Universal Robots PolyScope program: run_driver.urp

Program run_driver (installation=default directory=/programs/usbdisk/script_driver createdIn=5.2.0.61336 lastSavedIn=5.3.0.64176 robotSerialNumber=20195000535)
Calibrated DH parameters: a=[0.000149, -0.595503, -0.570094, 0.000069, 0.000037, 0]; d=[0.180711, 684.397239, -686.764447, 2.541569, 0.119967, 0.115293]; alpha=[1.570175, 0.000207, -0.013852, 1.571079, -1.570194, 0]; deltaTheta=[0, 0.233602, -0.176156, -0.057447, 0, 0]
BeforeStart
  Script file /programs/usbdisk/script_driver/driver.script
    | def driver():
    |   # Initialize variables hi
    |   global mode_thread_running = -1
    |   reset_vars()
    |   # Setup thread to read and update registers
    |   run read_and_update()
    |   # Continuously run command() function, which handles running correct mode thread. The mode threads then command the robot.
    |   while (True):
    |     command()
    |     sync()
    |   end
    | end
    | 
    | def command():
    |   # Run correct mode thread, then continuously check if the current thread is still running.
    |   # If mode switches while a mode thread is currently running, kill that mode thread
    |   # Break the loop and return from this function once either the mode thread finishes or the mode thread is killed
    |   mode_thread_switch() # Run the correct mode thread. This will update global variable mode_thread_running
    |   sync()
    |   while (mode_thread_running != -1): # mode_thread_running = mode number of mode thread that is currently running, otherwise if no mode thread is running, it = -1
    |     if mode != mode_thread_running: # If mode switched while another mode thread is already running, kill the current mode thread before breaking loop
    |       kill mode_thread_handler
    |       mode_thread_running = -1
    |     else:
    |       sync()
    |     end
    |   end
    | end
    | 
    | def mode_thread_switch():
    |   # Based on current value of mode, run the corresponding mode thread
    |   end_freedrive_mode() # End freedrive mode (if not in freedrive mode, does nothing) before running a mode thread
    |   if mode == STANDBY_MODE or enable == 0:
    |     global mode_thread_handler = run standby()
    |   elif mode == FREEDRIVE_MODE:
    |     global mode_thread_handler = run freedrive()
    |   elif mode == WAYPOINT_JOINT_MODE:
    |     global mode_thread_handler = run waypointJoint()
    |   elif mode == WAYPOINT_CARTESIAN_MODE:
    |     global mode_thread_handler = run waypointCartesian()
    |   elif mode == POSITION_CONTROL_JOINT_MODE:
    |     global mode_thread_handler = run posControlJoint()
    |   elif mode == POSITION_CONTROL_CARTESIAN_MODE:
    |     global mode_thread_handler = run posControlCartesian()
    |   elif mode == VELOCITY_CONTROL_JOINT_MODE:
    |     global mode_thread_handler = run velControlJoint()
    |   elif mode == VELOCITY_CONTROL_CARTESIAN_MODE:
    |     global mode_thread_handler = run velControlCartesian()
    |   end
    | end
    | 
    | thread read_and_update():
    |   # Continuously
    |   while(True):
    |     write_output_integer_register(PING_OUTPUT_INT_REGISTER, read_input_integer_register(PING_INT_REGISTER))
    |     if mode != read_input_integer_register(MODE_INT_REGISTER): # If mode changed, reset variables and re-setup watchdogs
    |       reset_vars()
    |       mode = read_input_integer_register(MODE_INT_REGISTER)
    |       setup_watchdogs()
    |     end
    |     # Update each variable only if mode requires it to be updated. Create list of all modes which require variable to be updated and use list_contains() to check if current mode is one of those modes
    |     if list_contains(mode, [WAYPOINT_JOINT_MODE, WAYPOINT_CARTESIAN_MODE, POSITION_CONTROL_JOINT_MODE, POSITION_CONTROL_CARTESIAN_MODE, VELOCITY_CONTROL_JOINT_MODE, VELOCITY_CONTROL_CARTESIAN_MODE]):
    |       setp = read_registers_into_list(SETP_DOUBLE_REGISTER_OFFSET, 6, "DOUBLE")
    |     end
    |     if list_contains(mode, [WAYPOINT_JOINT_MODE, WAYPOINT_CARTESIAN_MODE,VELOCITY_CONTROL_JOINT_MODE]):
    |       avtr = read_registers_into_list(AVTR_DOUBLE_REGISTER_OFFSET, 4, "DOUBLE")
    |     end
    |     if list_contains(mode, [POSITION_CONTROL_JOINT_MODE, POSITION_CONTROL_CARTESIAN_MODE, VELOCITY_CONTROL_CARTESIAN_MODE]):
    |       servoj_params = read_registers_into_list(SERVOJ_PARAMS_DOUBLE_REGISTER_OFFSET, 3, "DOUBLE")
    |     end
    |     enable = read_input_integer_register(ENABLE_INT_REGISTER) # Always update enable regardless of mode
    |     sync()
    |   end
    | end
    | 
    | def reset_vars():
    |   global mode = 0
    |   global enable = 0
    |   global setp = [0.0,0.0,0.0,0.0,0.0,0.0]
    |   global avtr = [0.0,0.0,0.0,0.0]
    |   global servoj_params = [0.0,0.0,0.0]
    | end
    | 
    | def setup_watchdogs():
    |   # Depending on current mode, set watchdog frequencies and responses for each watchdog
    |   # Right now, frequency always set to 500Hz and response is "STOP" if mode requires that variable, or "IGNORE" otherwise
    |   # "STOP" preferred over "PAUSE" initially for safety. Once we are more comfortable with system, can use "PAUSE" where appropriate
    | 
    |   mode_freq = 1
    |   enable_freq = 1
    |   setp_freq = 1
    |   avtr_freq = 1
    |   servoj_params_freq = 1
    | 
    |   mode_resp = "IGNORE"
    |   enable_resp = "IGNORE"
    |   setp_resp = "IGNORE"
    |   avtr_resp = "IGNORE"
    |   servoj_params_resp = "IGNORE"
    | 
    |   if list_contains(mode, [POSITION_CONTROL_JOINT_MODE, POSITION_CONTROL_CARTESIAN_MODE, VELOCITY_CONTROL_JOINT_MODE, VELOCITY_CONTROL_CARTESIAN_MODE, FORCE_CONTROL_MODE]):
    |     mode_resp = "STOP"
    |   end
    |   if list_contains(mode, [POSITION_CONTROL_JOINT_MODE, POSITION_CONTROL_CARTESIAN_MODE, VELOCITY_CONTROL_JOINT_MODE, VELOCITY_CONTROL_CARTESIAN_MODE, FORCE_CONTROL_MODE]):
    |     enable_resp = "STOP"
    |   end
    |   if list_contains(mode, [POSITION_CONTROL_JOINT_MODE, POSITION_CONTROL_CARTESIAN_MODE, VELOCITY_CONTROL_JOINT_MODE, VELOCITY_CONTROL_CARTESIAN_MODE, FORCE_CONTROL_MODE]):
    |     setp_resp = "STOP"
    |   end
    |   if list_contains(mode, []):
    |     avtr_resp = "STOP"
    |   end
    |   if list_contains(mode, [POSITION_CONTROL_JOINT_MODE, POSITION_CONTROL_CARTESIAN_MODE, VELOCITY_CONTROL_CARTESIAN_MODE]):
    |     servoj_params_resp = "STOP"
    |   end
    | 
    |   rtde_set_watchdog("input_int_register_"+to_str(MODE_INT_REGISTER), mode_freq, mode_resp)
    |   rtde_set_watchdog("input_int_register_"+to_str(ENABLE_INT_REGISTER), enable_freq, enable_resp)
    |   rtde_set_watchdog("input_double_register_"+to_str(SETP_DOUBLE_REGISTER_OFFSET), setp_freq, setp_resp)
    |   rtde_set_watchdog("input_double_register_"+to_str(AVTR_DOUBLE_REGISTER_OFFSET), avtr_freq, avtr_resp)
    |   rtde_set_watchdog("input_double_register_"+to_str(SERVOJ_PARAMS_DOUBLE_REGISTER_OFFSET), servoj_params_freq, servoj_params_resp)
    | end
    | 
    | 
    | # MODE THREADS
    | # FIRST set mode_thread_running to the corresponding mode number.
    | # THEN body of thread
    | thread standby():
    |   mode_thread_running = STANDBY_MODE
    |   write_output_integer_register(MODE_OUTPUT_INT_REGISTER, mode_thread_running)
    |   while(True):
    |     if not is_steady():
    |       stopj(DEFAULT_JOINT_ACCELERATION)
    |     end
    |     sync()
    |   end
    | end
    | 
    | thread freedrive():
    |   mode_thread_running = FREEDRIVE_MODE
    |   write_output_integer_register(MODE_OUTPUT_INT_REGISTER, mode_thread_running)
    | 
    |   if not is_steady():
    |     stopj(DEFAULT_JOINT_ACCELERATION)
    |   end
    |   freedrive_mode()
    |   # Loop inside this thread so freedrive() only gets called once instead of continuously. Necessary so that stopj() only called one time
    |   # Thread will be killed inside command() function once mode is switched to something other than freedrive mode
    |   while(True):
    |     sync()
    |   end
    | end
    | 
    | thread waypointJoint():
    |   mode_thread_running = WAYPOINT_JOINT_MODE
    |   write_output_integer_register(MODE_OUTPUT_INT_REGISTER, mode_thread_running)
    |   while(True):
    |     if not is_steady():
    |       stopj(DEFAULT_JOINT_ACCELERATION)
    |     end
    |     if not diff_norm_within_tol(setp, get_target_joint_positions(), 0.0001) and avtr[0] > 0 and avtr[1] > 0:
    |       movej(setp, avtr[0], avtr[1], avtr[2], avtr[3])
    |     end
    |     sync()
    |   end
    | end
    | 
    | thread waypointCartesian():
    |   # THIS MODE IS CURRENTLY VERY UNSTABLE. DO NOT USE UNLESS WAYPOINT IS CLOSE TO CURRENT POSITION
    |   # One way to make this more usable is to use movej instead of movel. We can still give the robot a cartesian position, but it will move there linearly in joint space
    |   # Possibly needs to be broken into sub-modes (waypointJointj, waypointJointl, waypointCartesianj, waypointCartesianl) where Joint vs Cartesian specifies which set point is used and the j vs l suffix specifies whether the path is linearly interpolated in joint space or cartesian space
    |   mode_thread_running = WAYPOINT_CARTESIAN_MODE
    |   write_output_integer_register(MODE_OUTPUT_INT_REGISTER, mode_thread_running)
    |   while(True):
    |     if not is_steady():
    |       stopj(DEFAULT_JOINT_ACCELERATION)
    |     end
    |     if not diff_norm_within_tol(setp, pose_to_list(get_target_tcp_pose()), 0.0001) and avtr[0] > 0 and avtr[1] > 0:
    |       movel(list_to_pose(setp), avtr[0], avtr[1], avtr[2], avtr[3])
    |     end
    |     sync()
    |   end
    | end
    | 
    | thread posControlJoint():
    |   mode_thread_running = POSITION_CONTROL_JOINT_MODE
    |   write_output_integer_register(MODE_OUTPUT_INT_REGISTER, mode_thread_running)
    |   while(True):
    |     servoj(setp, 0, 0, servoj_params[0], servoj_params[1], servoj_params[2])
    |     sync()
    |   end
    |   mode_thread_running = -1
    | end
    | 
    | thread posControlCartesian():
    |   mode_thread_running = POSITION_CONTROL_CARTESIAN_MODE
    |   write_output_integer_register(MODE_OUTPUT_INT_REGISTER, mode_thread_running)
    |   while(True):
    |     servoj(get_inverse_kin(list_to_pose(setp)), 0, 0, servoj_params[0], servoj_params[1], servoj_params[2])
    |     sync()
    |   end
    | end
    | 
    | thread velControlJoint():
    |   mode_thread_running = VELOCITY_CONTROL_JOINT_MODE
    |   write_output_integer_register(MODE_OUTPUT_INT_REGISTER, mode_thread_running)
    |   while(True):
    |     speedj(setp, avtr[0], avtr[2])
    |     #speedj(setp,5,0.01)
    | 
    |     sync()
    |   end
    | end
    | 
    | thread velControlCartesian():
    |   mode_thread_running = VELOCITY_CONTROL_CARTESIAN_MODE
    |   write_output_integer_register(MODE_OUTPUT_INT_REGISTER, mode_thread_running)
    |   Kp = [1.0,1.0,1.0,1.0,1.0,1.0]
    |   Ki = [0.0,0.0,0.0,0.0,0.0,0.0]
    |   err_i = [0.0,0.0,0.0,0.0,0.0,0.0]
    |   while(True):
    |     err = list_subtract(setp, pose_to_list(get_actual_tcp_speed()))
    |     err_i = list_add(err_i,err)
    |     p_term = list_multiply(Kp, err)
    |     i_term = list_multiply(Ki, err_i)
    | 
    |     pos_setp = list_add(pose_to_list(get_actual_tcp_pose()), list_add(p_term,i_term))
    | 
    |     servoj(get_inverse_kin(list_to_pose(pos_setp)), 0, 0, servoj_params[0], servoj_params[1], servoj_params[2])
    |     sync()
    |   end
    | end
    | 
    | thread forceControl():
    |   mode_thread_running = FORCE_CONTROL_MODE
    |   mode_thread_running = -1
    | end
  Script file /programs/usbdisk/script_driver/driver_helper_functions.script
    | # REGISTER INDICES/OFFSETS
    | MODE_INT_REGISTER = 0
    | ENABLE_INT_REGISTER = 1
    | PING_INT_REGISTER = 2
    | 
    | SETP_DOUBLE_REGISTER_OFFSET = 0
    | AVTR_DOUBLE_REGISTER_OFFSET = 6
    | SERVOJ_PARAMS_DOUBLE_REGISTER_OFFSET = 10
    | 
    | # MODE NUMBERS
    | STANDBY_MODE = 0
    | FREEDRIVE_MODE = 1
    | WAYPOINT_JOINT_MODE = 2
    | WAYPOINT_CARTESIAN_MODE = 3 # THIS MODE IS VERY UNSTABLE RIGHT NOW. RECOMMEND NOT USING UNLESS WAYPOINT IS RELATIVELY CLOSE TO CURRENT POSITION. FOR FAR AWAY WAYPOINTS, ROBOT WILL LIKELY RAISE ERROR AND STOP MOTION
    | POSITION_CONTROL_JOINT_MODE = 4
    | POSITION_CONTROL_CARTESIAN_MODE = 5
    | VELOCITY_CONTROL_JOINT_MODE = 6
    | VELOCITY_CONTROL_CARTESIAN_MODE = 7
    | FORCE_CONTROL_MODE = 8
    | 
    | MODE_OUTPUT_INT_REGISTER = 0
    | PING_OUTPUT_INT_REGISTER = 1
    | 
    | DEFAULT_JOINT_ACCELERATION = 1.4
    | 
    | def list_contains(value, list):
    |   # Checks if a list contains at least one element equal to "value". Returns True if so, False otherwise
    |   i = 0
    |   while i < length(list):
    |     if (list[i] == value):
    |       return True
    |     end
    |     i = i + 1
    |   end
    |   return False
    | end
    | 
    | def init_list(n, type):
    |   # Initializes and returns a list of size n. The elements of the list are of type "type"
    |   # type can be either "INT" or "DOUBLE". Right now, if any other value is passed for type, will crash because i not defined
    |   # n can be any integer between 1 and 6. Right now, if any other value is passed for n, will crash because list not defined
    |   if type == "INT":
    |     i = 0
    |   elif type == "DOUBLE":
    |     i = 0.0
    |   end
    |   if n == 1:
    |     list = [i]
    |   elif n == 2:
    |     list = [i,i]
    |   elif n == 3:
    |     list = [i,i,i]
    |   elif n == 4:
    |     list = [i,i,i,i]
    |   elif n == 5:
    |     list = [i,i,i,i,i]
    |   elif n == 6:
    |     list = [i,i,i,i,i,i]
    |   end
    |   return list
    | end
    | 
    | def list_to_pose(list):
    |   # Creates and returns a pose with the first 6 elements of "list". The values are copied directly (i.e. no kinematics or IK)
    |   # Right now, if length of "list" is less than 6, this function will crash
    |   pose = p[0.0,0.0,0.0,0.0,0.0,0.0]
    |   i = 0
    |   while i < 6:
    |     pose[i] = list[i]
    |     i = i + 1
    |   end
    |   return pose
    | end
    | 
    | def pose_to_list(pose):
    |   # Creates and returns a list with the first 6 elements of "pose". The values are copied directly (i.e. no kinematics or IK)
    |   # Right now, if length of "pose" is less than 6, this function will crash
    |   list = [0.0,0.0,0.0,0.0,0.0,0.0]
    |   i = 0
    |   while i < 6:
    |     list[i] = pose[i]
    |     i = i + 1
    |   end
    |   return list
    | end
    | 
    | def diff_norm_within_tol(list1, list2, tol):
    |   # Returns true if Euclidian norm of difference between list1 and list2 is <= tolerance "tol"
    |   # Used mostly to determine if two 6-DOF vectors/lists are "close enough"
    |   return norm(list_subtract(list1, list2)) <= tol
    | end
    | 
    | def read_registers_into_list(first, n, type):
    |   # reads n registers consecutively starting with register with index "first". "type" indicates the register type. "INT" -> integer_register, "DOUBLE" -> float_register
    |   # Example: read_registers_into_list(first=2, n=3, type="DOUBLE") -> return list: [input_float_register_2, input_float_register_3, input_float_register_4]
    |   # Right now, supports only "INT" and "DOUBLE" types
    |   list = init_list(n,type)
    |   i = 0
    |   while i < n:
    |     if type == "INT":
    |       list[i] = read_input_integer_register(first + i)
    |     elif type == "DOUBLE":
    |       list[i] = read_input_float_register(first + i)
    |     end
    |     i = i + 1
    |   end
    |   return list
    | end
    | 
    | def min(a,b):
    |   if a < b:
    |     return a
    |   else:
    |     return b
    |   end
    | end
    | 
    | def max(a,b):
    |   if a > b:
    |     return a
    |   else:
    |     return b
    |   end
    | end
    | 
    | def list_subtract(list1, list2):
    |   # Subtract 2 lists element-wise (list1 - list2). The first n list elements are subtracted, where n is the length of the shortest list. The returned result is a list of length n
    |   # If shortest list has length < 1 or length > 6, function init_list() will crash
    |   n = min(length(list1), length(list2))
    |   result = init_list(n, "DOUBLE")
    |   i = 0
    |   while i < n:
    |     result[i] = list1[i]-list2[i]
    |     i = i + 1
    |   end
    |   return result
    | end
    | 
    | def list_add(list1, list2):
    |   # Add 2 lists element-wise. The first n list elements are subtracted, where n is the length of the shortest list. The returned result is a list of length n
    |   # If shortest list has length < 1 or length > 6, function init_list() will crash
    |   n = min(length(list1), length(list2))
    |   result = init_list(n, "DOUBLE")
    |   i = 0
    |   while i < n:
    |     result[i] = list1[i]+list2[i]
    |     i = i + 1
    |   end
    |   return result
    | end
    | 
    | def list_multiply(list1, list2):
    |   # Multiply 2 lists element-wise. The first n list elements are multiplied, where n is the length of the shortest list. The returned result is a list of length n
    |   # If shortest list has length < 1 or length > 6, function init_list() will crash
    |   n = min(length(list1), length(list2))
    |   result = init_list(n, "DOUBLE")
    |   i = 0
    |   while i < n:
    |     result[i] = list1[i]*list2[i]
    |     i = i + 1
    |   end
    |   return result
    | end
Robot Program (runOnlyOnce=true)
  Script: driver()
